{attribute 'OPC.UA.DA.StructuredType' := '1'}
FUNCTION_BLOCK FB_UVFilter_Pentair_EU40 EXTENDS FB_BaseDevice IMPLEMENTS I_Device

VAR
	{attribute 'OPC.UA.DA' := '1'} 
	bInRelay AT %I*: BOOL := FALSE;
	
	{attribute 'OPC.UA.DA' := '1'} 
	bOutRelay AT %Q*: BOOL := FALSE;
	
	{attribute 'OPC.UA.DA' := '0'} 
	eSMState: (WAIT, TURNING_ON, ON, TURNING_OFF, OFF);
	
	{attribute 'OPC.UA.DA' := '0'} 
	tActionTimeout: TIME := T#5S;
	{attribute 'OPC.UA.DA' := '0'} 
	fbTON_timeout: TON := (PT := tActionTimeout, IN := FALSE);
END_VAR

IF GVL.bAutoUpdateDeviceState THEN
	eState := eStateTarget;	
END_IF

IF eMode = E_DeviceMode.MANUAL THEN
	bEnable := TRUE;
END_IF

IF (eStateTarget = E_DeviceState.ON) AND bEnable AND eSMState <> ON THEN
	eSMState := TURNING_ON;
END_IF

IF ((eStateTarget = E_DeviceState.OFF) OR (NOT bEnable)) AND eSMState <> OFF THEN
	eSMState := TURNING_OFF;
END_IF



CASE eSMState OF
	
		
	TURNING_ON: 
		bOutRelay := TRUE;
		eSMState := ON;
		eState := E_DeviceState.ON;
		
	ON:
		IF NOT bOutRelay THEN
			eSMState := TURNING_OFF;
		END_IF
		
	TURNING_OFF:
		bOutRelay := FALSE;
		eSMState := OFF;
		eState := E_DeviceState.TURNING_OFF;
		
	OFF:
		eState := E_DeviceState.OFF;
		bBusy := FALSE;
		
END_CASE

{warning 'add method implementation '}
METHOD disable : BOOL
bEnable := FALSE;
END_METHOD

{warning 'add method implementation '}
METHOD enable : BOOL
bEnable := TRUE;
END_METHOD

METHOD FB_init : BOOL
VAR_INPUT
	bInitRetains : BOOL; // if TRUE, the retain variables are initialized (warm start / cold start)
	bInCopyCode : BOOL;  // if TRUE, the instance afterwards gets moved into the copy code (online change)
	
	UnitID: STRING(80);
	UnitDescr: STRING(255); 
END_VAR
sID := UnitID;
sDescr := UnitDescr;
END_METHOD

METHOD setOff : BOOL
VAR_INPUT
END_VAR
IF bEnable THEN
	eSMState := TURNING_OFF;
END_IF
END_METHOD

METHOD setOn : BOOL
VAR_INPUT
END_VAR
IF bEnable THEN
	eSMState := TURNING_ON;
END_IF
END_METHOD

END_FUNCTION_BLOCK

(* stored: Version 1.1.0.1, ProductVersion 3.1.4024.12
   POU FB_UVFilter_Pentair_EU40: Id {66450e10-72f9-4f09-98e9-94012e816dbf}, SpecialFunc None
   Method disable: Id {26ea0b53-814a-4abe-a4f6-3680a851d335}
   Method enable: Id {fca10751-3609-47b2-992a-a93960b24ef3}
   Method FB_init: Id {0a9c7970-3b42-4214-88e5-4d3a1acb1be8}
   Method setOff: Id {a49c8c7e-1503-4a0a-9631-50a15a090bf6}
   Method setOn: Id {89d75852-f0e4-4993-850f-a89750075b03} *)
